(* IEC 61131-3 sources: 83616---Application-of-Mechatronic-Systems---PROJECT/txt_export/Device.dev/Plc Logic/Application, 8 files *)

(* ---- BikeType.dut ---- *)
(*#-#-#-#-#-#-#-#-#-#---Declaration---#-#-#-#-#-#-#-#-#-#-#-#-#*)

{attribute 'qualified_only'}
{attribute 'to_string'}

TYPE BikeType :
(
	BMX := 1,
	Electric,
	Folding,
	Road
)DINT:=BMX;
END_TYPE

(* ---- eAccessories.dut ---- *)
(*#-#-#-#-#-#-#-#-#-#---Declaration---#-#-#-#-#-#-#-#-#-#-#-#-#*)

{attribute 'qualified_only'}
{attribute 'to_string'}
TYPE eAccessories :
(
	GPS := 1,
	Lights,
	Bell,
	Lock,
	Speedometer,
	None
)DINT:=GPS;
END_TYPE

(* ---- typ_accStats.dut ---- *)
(*#-#-#-#-#-#-#-#-#-#---Declaration---#-#-#-#-#-#-#-#-#-#-#-#-#*)

TYPE typ_accStats :
STRUCT
	uiGPS:UINT;
	uiLights:UINT;
	uiBell:UINT;
	uiLock:UINT;
	uiSpeedo:UINT;
END_STRUCT
END_TYPE

(* ---- typ_OrderData.dut ---- *)
(*#-#-#-#-#-#-#-#-#-#---Declaration---#-#-#-#-#-#-#-#-#-#-#-#-#*)

TYPE typ_OrderData :
STRUCT
	ulOrderNo: INT := 0;
	uiQty: INT;
	eType: STRING;
	aeAccessories: ARRAY [1..4] OF STRING;
	status: STRING:='NA';
	asmLine: STRING:='NA';
END_STRUCT
END_TYPE

(* ---- GVL.gvl ---- *)
(*#-#-#-#-#-#-#-#-#-#---Declaration---#-#-#-#-#-#-#-#-#-#-#-#-#*)

{attribute 'qualified_only'}
VAR_GLOBAL
	OPCUA_Server: FB_OPCUA_Server;
END_VAR

(* ---- FB_OPCUA_Server.pou ---- *)
(*#-#-#-#-#-#-#-#-#-#---Declaration---#-#-#-#-#-#-#-#-#-#-#-#-#*)

FUNCTION_BLOCK FB_OPCUA_Server
VAR_INPUT
END_VAR
VAR_OUTPUT
	orderData: typ_OrderData;
END_VAR
VAR
END_VAR

(*#-#-#-#-#-#-#-#-#-#---Implementation---#-#-#-#-#-#-#-#-#-#-#-#-#*)

(* ---- RANDI.pou ---- *)
(*#-#-#-#-#-#-#-#-#-#---Declaration---#-#-#-#-#-#-#-#-#-#-#-#-#*)

FUNCTION_BLOCK RANDI
VAR_INPUT
END_VAR
VAR_OUTPUT
	di_Result: DINT;
END_VAR
VAR
	X:DINT:=23;
	A:DINT:=47;
	M:DINT:=100;
	B:DINT:=11;
	ARR: ARRAY [1..100] OF INT:=[4  , 4   ,6   ,2   ,2   ,1   ,6   ,4   ,3   ,4   ,4   ,4   ,4   ,5   ,4   ,6   ,2   ,1   ,1   ,1   ,3   ,3   ,3   ,5   ,4   ,5 ,6   ,6   ,2   ,1   ,5  , 1   ,4   ,4   ,6   ,3   ,3   ,5   ,5   ,4   ,3   ,1   ,4   ,2   ,1   ,5   ,2   ,3   ,5   ,3   ,5  , 3 ,5   ,5   ,3   ,1   ,2   ,3   ,2   ,2   ,5   ,3   ,6   ,3   ,5  , 3   ,5   ,5   ,3   ,2   ,5   ,6   ,2   ,5   ,3   ,6   ,5   ,2 ,6   ,6   ,4   ,6   ,4   ,1   ,2   ,3   ,5   ,5   ,5   ,2   ,4   ,1   ,1   ,1   ,5   ,3   ,2   ,3   ,1   ,1];
	ARR1: ARRAY[1..1] OF DINT:=[0];
END_VAR

(*#-#-#-#-#-#-#-#-#-#---Implementation---#-#-#-#-#-#-#-#-#-#-#-#-#*)

X:=((X*A)+B) MOD M;
IF X=ARR1[1] THEN
	X:=((X*A)+B) MOD M;
	di_Result:=ARR[X];
ELSE
	di_Result:=ARR[X];
	ARR1[1]:=X;
END_IF

(* ---- PLC_PRG.pou ---- *)
(*#-#-#-#-#-#-#-#-#-#---Declaration---#-#-#-#-#-#-#-#-#-#-#-#-#*)

PROGRAM PLC_PRG
VAR
fbWebServer:FB_WebServer;
fbAssemblyLine:ARRAY [0..4] OF FB_AssemblyLine;
fbAssemblyAdd: ARRAY[0..4] OF POINTER TO fb_AssemblyLine :=	[ADR(fbAssemblyLine[0]),
																 ADR(fbAssemblyLine[1]),
																 ADR(fbAssemblyLine[2]),
																 ADR(fbAssemblyLine[3]),
																 ADR(fbAssemblyLine[4])];
fbOrderParser: FB_OrderParser(pFB_Server := ADR(fbWebServer),apFB_AssemblyLine:=fbAssemblyAdd);
i:INT;
fb_Ass: FB_AssemblyLine;
assem_line:INT;
assembly_line: ARRAY [0..4] OF STRING:=['ASSEMBLY_LINE_0','ASSEMBLY_LINE_1','ASSEMBLY_LINE_2','ASSEMBLY_LINE_3','ASSEMBLY_LINE_4'];
Web_Visu: ARRAY [1..3] OF STRING:=['HMI_ORDER','Visu_Order','Visu_Assembly_Display'];
web: INT;

END_VAR
(*#-#-#-#-#-#-#-#-#-#---Implementation---#-#-#-#-#-#-#-#-#-#-#-#-#*)

fbWebServer(); //simulate web orders
fbOrderParser();
FOR I:=0 TO 4 BY 1 DO
	fbAssemblyLine[i]();
END_FOR
IF web=1 THEN
	CurrentVisu:='HMI_ORDER';
ELSIF web=2 THEN
	CurrentVisu:='Visu_Order';
ELSIF web=3 THEN
	CurrentVisu:='Visu_Assembly_Display';
END_IF
IF assem_line=0 THEN
	fb_Ass:=fbAssemblyLine[0];
ELSIF assem_line=1 THEN
	fb_Ass:=fbAssemblyLine[1];
ELSIF assem_line=2 THEN
	fb_Ass:=fbAssemblyLine[2];
ELSIF assem_line=3 THEN
	fb_Ass:=fbAssemblyLine[3];
ELSIF assem_line=4 THEN
	fb_Ass:=fbAssemblyLine[4];
END_IF
